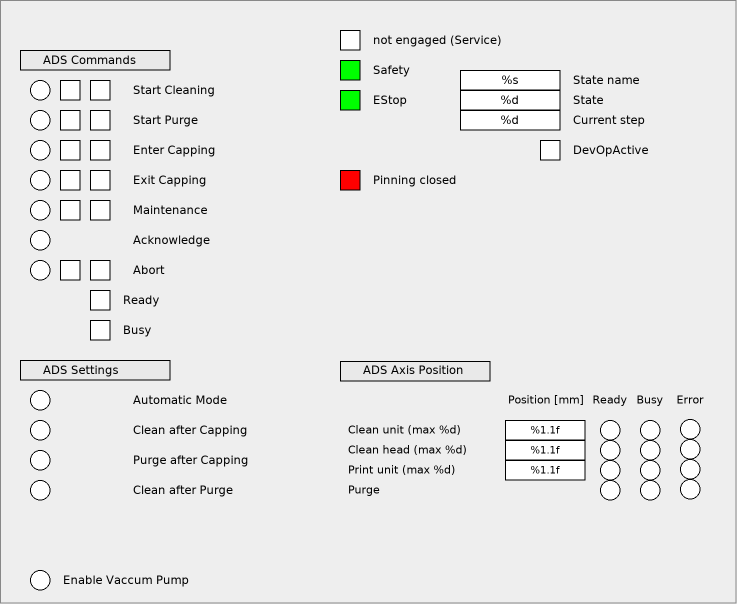
VISUALIZATION _VISU_CLEAN_PROCESS  // 737x604
VAR_IN_OUT
  m_Inst : INT;               (*visu instance*) 
END_VAR
    Rectangle (0,0 737x604)
    Polyline (20,50)
    Polyline (360,360)
    Rectangle (130,80 90x20), "Start Cleaning"
    Ellipse (30,80 20x20), colour toggle: PRG_MACHINE.sADS_CleanProcess[m_Inst].bI_Clean
        tap PRG_MACHINE.sADS_CleanProcess[m_Inst].bI_Clean
    Rectangle (130,110 90x20), "Start Purge"
    Rectangle (130,140 90x20), "Enter Capping"
    Rectangle (130,170 90x20), "Exit Capping"
    Rectangle (130,200 90x20), "Maintenance"
    RoundedRectangle (90,290 20x20), colour toggle: PRG_MACHINE.sADS_CleanProcess[m_Inst].bO_Ready
    Rectangle (120,290 120x20), "Ready"
    Rectangle (460,70 100x20), "%s", text variable: PRG_MACHINE.fb_CleanProcess[m_Inst].sL_CurrentState^.sL_StateName
    Rectangle (570,70 100x20), "State name"
    Rectangle (460,90 100x20), "%d", text variable: PRG_MACHINE.fb_CleanProcess[m_Inst].sL_CurrentState^.iL_State
    Rectangle (570,90 100x20), "State"
    Rectangle (20,50 150x20)
    Rectangle (40,50 130x20), "ADS Commands"
    RoundedRectangle (60,80 20x20), colour toggle: PRG_MACHINE.sADS_CleanProcess[m_Inst].bO_CleanCanEx
    RoundedRectangle (90,80 20x20), colour toggle: PRG_MACHINE.sADS_CleanProcess[m_Inst].bO_CleanExec
    Ellipse (30,110 20x20), colour toggle: PRG_MACHINE.sADS_CleanProcess[m_Inst].bI_Purge
        tap PRG_MACHINE.sADS_CleanProcess[m_Inst].bI_Purge
    RoundedRectangle (60,110 20x20), colour toggle: PRG_MACHINE.sADS_CleanProcess[m_Inst].bO_PurgeCanEx
    RoundedRectangle (90,110 20x20), colour toggle: PRG_MACHINE.sADS_CleanProcess[m_Inst].bO_PurgeExec
    Ellipse (30,140 20x20), colour toggle: PRG_MACHINE.sADS_CleanProcess[m_Inst].bI_StartCapping
        tap PRG_MACHINE.sADS_CleanProcess[m_Inst].bI_StartCapping
    RoundedRectangle (60,140 20x20), colour toggle: PRG_MACHINE.sADS_CleanProcess[m_Inst].bO_StartCappingCanEx
    RoundedRectangle (90,140 20x20), colour toggle: PRG_MACHINE.sADS_CleanProcess[m_Inst].bO_StartCappingExec
    Ellipse (30,170 20x20), colour toggle: PRG_MACHINE.sADS_CleanProcess[m_Inst].bI_StopCapping
        tap PRG_MACHINE.sADS_CleanProcess[m_Inst].bI_StopCapping
    RoundedRectangle (60,170 20x20), colour toggle: PRG_MACHINE.sADS_CleanProcess[m_Inst].bO_StopCappingCanEx
    RoundedRectangle (90,170 20x20), colour toggle: PRG_MACHINE.sADS_CleanProcess[m_Inst].bO_StopCappingExec
    Ellipse (30,200 20x20), colour toggle: PRG_MACHINE.sADS_CleanProcess[m_Inst].bI_Maintenance
        tap PRG_MACHINE.sADS_CleanProcess[m_Inst].bI_Maintenance
    RoundedRectangle (60,200 20x20), colour toggle: PRG_MACHINE.sADS_CleanProcess[m_Inst].bO_MaintenanceCanEx
    RoundedRectangle (90,200 20x20), colour toggle: PRG_MACHINE.sADS_CleanProcess[m_Inst].bO_MaintenanceExec
    Rectangle (130,260 90x20), "Abort"
    Ellipse (30,260 20x20), colour toggle: PRG_MACHINE.sADS_CleanProcess[m_Inst].bI_Abort
        tap PRG_MACHINE.sADS_CleanProcess[m_Inst].bI_Abort
    RoundedRectangle (60,260 20x20), colour toggle: PRG_MACHINE.sADS_CleanProcess[m_Inst].bO_AbortCanEx
    RoundedRectangle (90,260 20x20), colour toggle: PRG_MACHINE.sADS_CleanProcess[m_Inst].bO_AbortExec
    RoundedRectangle (90,320 20x20), colour toggle: PRG_MACHINE.sADS_CleanProcess[m_Inst].bO_Busy
    Rectangle (120,320 120x20), "Busy"
    Rectangle (20,360 150x20)
    Rectangle (40,360 130x20), "ADS Settings"
    Polyline (40,360)
    RoundedRectangle (340,90 20x20), colour toggle: NOT PRG_MACHINE.bL_IO_EStopOK
    Rectangle (370,30 180x20), "not engaged (Service)"
    Rectangle (505,420 80x20), "%1.1f", text variable: PRG_MACHINE.sADS_CleanAxis[iCPr_MAP_Cp_CuAxis[m_Inst]].sO_AxisPosition.fO_Val
    Rectangle (505,440 80x20), "%1.1f", text variable: PRG_MACHINE.sADS_CleanAxis[iCPr_MAP_Cp_ChAxis[m_Inst]].sO_AxisPosition.fO_Val
    Rectangle (505,460 80x20), "%1.1f", text variable: PRG_MACHINE.sADS_CleanAxis[iCPr_MAP_Cp_PuAxis[m_Inst]].sO_AxisPosition.fO_Val
    Ellipse (600,420 20x20), colour toggle: PRG_MACHINE.sADS_CleanAxis[iCPr_MAP_Cp_CuAxis[m_Inst]].bO_Ready
    Ellipse (640,420 20x20), colour toggle: PRG_MACHINE.sADS_CleanAxis[iCPr_MAP_Cp_CuAxis[m_Inst]].bO_Busy
    Ellipse (600,440 20x20), colour toggle: PRG_MACHINE.sADS_CleanAxis[iCPr_MAP_Cp_ChAxis[m_Inst]].bO_Ready
    Ellipse (640,440 20x20), colour toggle: PRG_MACHINE.sADS_CleanAxis[iCPr_MAP_Cp_ChAxis[m_Inst]].bO_Busy
    Ellipse (600,460 20x20), colour toggle: PRG_MACHINE.sADS_CleanAxis[iCPr_MAP_Cp_PuAxis[m_Inst]].bO_Ready
    Ellipse (640,460 20x20), colour toggle: PRG_MACHINE.sADS_CleanAxis[iCPr_MAP_Cp_PuAxis[m_Inst]].bO_Busy
    Rectangle (590,390 40x20), "Ready"
    Rectangle (630,390 40x20), "Busy"
    Rectangle (505,390 83x20), "Position [mm]"
    Rectangle (340,361 150x20)
    Rectangle (360,360 130x20), "ADS Axis Position"
    Ellipse (600,480 20x20), colour toggle: PRG_MACHINE.sADS_CleanAxis[iCPr_MAP_Cp_InkInterface[m_Inst]].bO_Ready
    Ellipse (640,480 20x20), colour toggle: PRG_MACHINE.sADS_CleanAxis[iCPr_MAP_Cp_InkInterface[m_Inst]].bO_Busy
    Rectangle (345,480 150x20), "Purge"
    Ellipse (680,419 20x20), colour toggle: PRG_MACHINE.sADS_CleanAxis[iCPr_MAP_Cp_CuAxis[m_Inst]].bO_Error
        toggle PRG_MACHINE.sADS_CleanAxis[iCPr_MAP_Cp_CuAxis[m_Inst]].bI_FaultAck
    Ellipse (680,439 20x20), colour toggle: PRG_MACHINE.sADS_CleanAxis[iCPr_MAP_Cp_ChAxis[m_Inst]].bO_Error
        toggle PRG_MACHINE.sADS_CleanAxis[iCPr_MAP_Cp_ChAxis[m_Inst]].bI_FaultAck
    Ellipse (680,459 20x20), colour toggle: PRG_MACHINE.sADS_CleanAxis[iCPr_MAP_Cp_PuAxis[m_Inst]].bO_Error
        tap PRG_MACHINE.sADS_CleanAxis[iCPr_MAP_Cp_PuAxis[m_Inst]].bI_FaultAck
    Rectangle (670,390 40x20), "Error"
    Ellipse (680,479 20x20), colour toggle: PRG_MACHINE.sADS_CleanAxis[iCPr_MAP_Cp_InkInterface[m_Inst]].bO_Error
    RoundedRectangle (340,60 20x20), colour toggle: NOT PRG_MACHINE.bL_SafetyOk[m_Inst]
    RoundedRectangle (340,30 20x20), colour toggle: PRG_MACHINE.fb_CleanProcess[m_Inst].bI_UsrService
    Rectangle (370,60 80x20), "Safety"
    Rectangle (370,90 80x20), "EStop"
    Rectangle (345,420 150x20), "Clean unit (max %d)", text variable: PRG_MACHINE.sADS_CleanAxis[iCPr_MAP_Cp_CuAxis[m_Inst]].sO_AxisPosition.fC_Max
    Rectangle (345,440 150x20), "Clean head (max %d)", text variable: PRG_MACHINE.sADS_CleanAxis[iCPr_MAP_Cp_ChAxis[m_Inst]].sO_AxisPosition.fC_Max
    Rectangle (345,460 150x20), "Print unit (max %d)", text variable: PRG_MACHINE.sADS_CleanAxis[iCPr_MAP_Cp_PuAxis[m_Inst]].sO_AxisPosition.fC_Max
    Rectangle (460,110 100x20), "%d", text variable: PRG_MACHINE.fb_CleanProcess[m_Inst].sL_CurrentState^.iL_State
    Rectangle (570,110 100x20), "Current step"
    RoundedRectangle (540,140 20x20), colour toggle: PRG_MACHINE.fb_CleanProcess[m_Inst].sL_CurrentState^.bL_DevOpActive
    Rectangle (570,140 100x20), "DevOpActive"
    Rectangle (130,390 103x20), "Automatic Mode"
    Ellipse (30,390 20x20), colour toggle: PRG_MACHINE.sADS_CleanProcess[m_Inst].bI_AutoMode
        toggle PRG_MACHINE.sADS_CleanProcess[m_Inst].bI_AutoMode
    Rectangle (130,420 150x20), "Clean after Capping"
    Ellipse (30,420 20x20), colour toggle: PRG_MACHINE.sADS_CleanProcess[m_Inst].bI_CleanAfterCapp
        toggle PRG_MACHINE.sADS_CleanProcess[m_Inst].bI_CleanAfterCapp
    Rectangle (130,480 150x20), "Clean after Purge"
    Ellipse (30,480 20x20), colour toggle: PRG_MACHINE.sADS_CleanProcess[m_Inst].bI_CleanAfterPurge
        toggle PRG_MACHINE.sADS_CleanProcess[m_Inst].bI_CleanAfterPurge
    Rectangle (130,450 150x20), "Purge after Capping"
    Ellipse (30,450 20x20), colour toggle: PRG_MACHINE.sADS_CleanProcess[m_Inst].bI_PurgeAfterCapp
        toggle PRG_MACHINE.sADS_CleanProcess[m_Inst].bI_PurgeAfterCapp
    Ellipse (30,570 20x20), colour toggle: PRG_MACHINE.bL_ManualVacuumBin[m_Inst]
        toggle PRG_MACHINE.bL_ManualVacuumBin[m_Inst]
    Rectangle (60,570 138x20), "Enable Vaccum Pump"
    RoundedRectangle (340,170 20x20), colour toggle: PRG_MACHINE.IbEAP_PinningClosed[m_Inst]
    Rectangle (370,170 150x20), "Pinning closed"
    Rectangle (130,230 90x20), "Acknowledge"
    Ellipse (30,230 20x20), colour toggle: PRG_MACHINE.sADS_CleanProcess[m_Inst].bI_Maintenance
        tap PRG_MACHINE.sADS_CleanProcess[m_Inst].bI_AcknowledgeError
END_VISUALIZATION

(* stored: Version 1.1.0.1, ProductVersion 3.1.4024.9
   Visu _VISU_CLEAN_PROCESS: Id {84c1126e-a0a2-46b1-a8f0-f5e111ab91ca} *)
